FUNCTION_BLOCK Q_SoftKeyMask (* Command change soft key mask( Part 6 - F.36 ) *)
  (* Standard: ISO 11783-6; Description: This command is used to change the soft key mask associated with a data or alarm mask object. Return values iso_s16 - E_NO_ERR ( 0 )  - OK - E_OVERFLOW (-6 ) - buffer overflow - E_NOACT (-8 ) - Command not possible in current state - E_NO_INSTANCE (-21) - No VT client available *)
  (* Version 1.0, 2022-07-08, franz *)
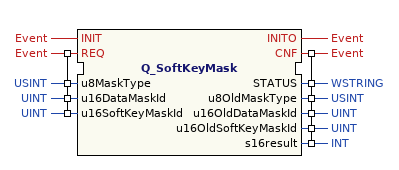
  EVENT_INPUT
    INIT; (* Service Initialization *)
    REQ WITH u16DataMaskId, u16SoftKeyMaskId, u8MaskType; (* Service Request *)
  END_EVENT
  EVENT_OUTPUT
    INITO; (* Initialization Confirm *)
    CNF WITH STATUS, s16result, u16OldDataMaskId, u16OldSoftKeyMaskId, u8OldMaskType; (* Confirmation of Requested Service *)
  END_EVENT
  VAR_INPUT
    u8MaskType : USINT; (* 1 == Data, 2 == Alarm *)
    u16DataMaskId : UINT; (* Object ID of active Mask *)
    u16SoftKeyMaskId : UINT; (* Object ID of (new) soft key mask *)
  END_VAR
  VAR_OUTPUT
    STATUS : WSTRING; (* Service Status *)
    u8OldMaskType : USINT;
    u16OldDataMaskId : UINT; (* Old object ID of active Mask *)
    u16OldSoftKeyMaskId : UINT; (* Old object ID of (new) soft key mask *)
    s16result : INT; (* retval see description *)
  END_VAR
END_FUNCTION_BLOCK
